# B&R Automation Studio project PP500_1
Automation Studio 4.12.3.127 SP; technology packages: mappCockpit 5.22.0, mappMotion 5.22.0, mappView 5.22.0

## Configuration PP500

CPU 5PP5CP.US15-02, AutomationRuntime F4.83, Build 4.1.2, Safety 1.10, Vc 

### Task classes (Cpu.sw)
```
Cyclic#8 (cycle 9600 us):
  Axis_1 <- Axis_1.prg
  Axis_2 <- Axis_2.prg
DataObjects: McAcpSys
NcDataObjects: McDriveLog
Binaries: arsvcreg, udbdef, mvLoader, McAcpDrv, arflatprv, arcoal, FWRules, TCData, mCoWebSc, McAcpSim, Config_1, ashwac, Settings, User, sysconf, iomap, asfw, arconfig, ashwd, Role, Config_2
Libraries: McBase, MpAxis, McAxis, MpBase, McAcpAx, CoTrace, AsZip, FileIO, runtime, AsSafety, standard, DataObj, AsXml, astime, AsBrStr, arssl, powerlnk, sys_lib, asepl, asieccon
```

### Hardware
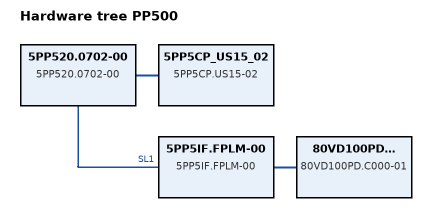
```
5PP520.0702-00 : 5PP520.0702-00 v2.1.3.1
  Connector IF3:
    ActivateDevice = 1
    ActivateSnmp = 2
5PP5CP_US15_02 : 5PP5CP.US15-02 v2.1.6.0  [SY -> 5PP520.0702-00.SY1]
  ConfigurationID = PP500_1_PP500
  UserPartitionSize = 64
  EnableUsbRemoteInstall = 1
  TimerDeviceType = EPLX2X
  TimerDevice = 5PP5IF.FPLM-00.IF1
  TaskClassIdleTime = 1600
  Cyclic1Duration = 800
  Cyclic1Tolerance = 800
  Cyclic3Duration = 40000
  Cyclic3Tolerance = 40000
  Cyclic8Duration = 9600
  FileDevice1
  FileDeviceName1 = USER
  FileDevicePath1 = USER_PATH
  ActivateOpcUa = 1
  OpcUaInformationModels_PV_Version = 1
5PP5IF.FPLM-00 : 5PP5IF.FPLM-00 v2.5.0.0  [SL -> 5PP520.0702-00.SL1]
  Connector IF1:
    CycleTime = 800
80VD100PD.C000-01 : 80VD100PD.C000-01 v2.5.0.0  [PLK1 -> 5PP5IF.FPLM-00.IF1 (NodeNumber=3) [Cable Type=PowerlinkCable, Length=10, Version=1.0.0.3]]
  DriveConfiguration/Module:
    McAcoposTypeID = AcoposMicroDConfig
    ActivateACOPOSSimulationOnPLC = 0
  DriveConfiguration/Channel[1]/RealAxis:
    AxisReference = gAxis_1
    MechanicalElementsIsInvisible = 0
  DriveConfiguration/Channel[1]/RealAxis/MechanicalElements/Gearbox:
    InputIsReadOnly = 0
    Input = 10
    OutputIsReadOnly = 0
    Output = 1
  DriveConfiguration/Channel[1]/RealAxis/MechanicalElements/RotaryToLinearTransformation:
    ReferenceDistanceIsReadOnly = 0
    ReferenceDistance = 36000
  DriveConfiguration/Channel[1]/RealAxis/Controller:
    ModeIsReadOnly = 0
    Mode = PositionControllerWithTorqueFeedForward
  DriveConfiguration/Channel[1]/RealAxis/Controller/Mode/Position:
    ProportionalGainIsReadOnly = 0
    ProportionalGain = 300
    IntegrationTimeIsReadOnly = 0
    IntegrationTime = 0.0
    TotalDelayTime = 0.0004
  DriveConfiguration/Channel[1]/RealAxis/Controller/Mode/Speed:
    ProportionalGainIsReadOnly = 0
    ProportionalGain = 0.4
    IntegrationTimeIsReadOnly = 0
    IntegrationTime = 0.0
    FilterTimeIsReadOnly = 0
    FilterTime = 0.0
  DriveConfiguration/Channel[1]/RealAxis/Controller/Mode:
    FeedForwardIsReadOnly = 0
    FeedForward = Standard
  DriveConfiguration/Channel[1]/RealAxis/Controller/Mode/FeedForward:
    TorqueLoad = 0.0
    TorquePositive = 0.016000
    TorqueNegative = 0.0
    SpeedTorqueFactor = 0.000300
    Inertia = 0.0
    AccelerationFilterTime = 0.0
  DriveConfiguration/Channel[1]/RealAxis/Controller/Mode/LoopFilters:
    LoopFilterXIsReadOnly = 0
    LoopFilter1 = NotUsed
    LoopFilter2 = NotUsed
    LoopFilter3 = NotUsed
  DriveConfiguration/Channel[1]/RealAxis/Homing:
    ModeIsReadOnly = 0
    Mode = Direct
  DriveConfiguration/Channel[1]/RealAxis/Homing/Mode:
    Position = 0.0
    ReferencePulse = NotUsed
  DriveConfiguration/Channel[1]/RealAxis/Homing:
    RestorePositionVariable = 
  DriveConfiguration/Channel[1]/RealAxis/StopReaction:
    QuickstopIsReadOnly = 0
    Quickstop = DecelerationLimit
    DriveErrorIsReadOnly = 0
    DriveError = DecelerationLimit
  DriveConfiguration/Channel[1]/RealAxis/MovementErrorLimits:
    PositionError = 10
    VelocityErrorMonitoring = Automatic1
  DriveConfiguration/Channel[1]/RealAxis:
    JerkFilterIsReadOnly = 0
    JerkFilter = NotUsed
    ZeroVibrationFilter = NotUsed
  DriveConfiguration/Channel[1]/RealAxis/DigitalInputs/HomingSwitch:
    SourceIsReadOnly = 0
    Source = NotUsed
    Level = High
  DriveConfiguration/Channel[1]/RealAxis/DigitalInputs/PositiveLimitSwitch:
    SourceIsReadOnly = 0
    Source = NotUsed
    Level = High
  DriveConfiguration/Channel[1]/RealAxis/DigitalInputs/NegativeLimitSwitch:
    SourceIsReadOnly = 0
    Source = NotUsed
    Level = High
  DriveConfiguration/Channel[1]/RealAxis/DigitalInputs/Trigger1:
    Source = X2Trigger1
    Level = High
  DriveConfiguration/Channel[1]/RealAxis/DigitalInputs/Trigger2:
    Source = X2Trigger2
    Level = High
  DriveConfiguration/Channel[1]/RealAxis/DigitalInputs/Quickstop:
    Input = Trigger2
  DriveConfiguration/Channel[1]/RealAxis/Simulation:
    SimulationModeOnPLC = SetValueGeneration
    SimulationModeOnACOPOS = NotUsed
  DriveConfiguration/Channel[1]/RealAxis/AxisFeatures:
    FeatureRef[1] = AxFeatureBrake
  DriveConfiguration/Channel[2]/RealAxis:
    AxisReference = gAxis_2
    MechanicalElementsIsInvisible = 0
  DriveConfiguration/Channel[2]/RealAxis/MechanicalElements/Gearbox:
    InputIsReadOnly = 0
    Input = 1
    OutputIsReadOnly = 0
    Output = 1
  DriveConfiguration/Channel[2]/RealAxis/MechanicalElements/RotaryToLinearTransformation:
    ReferenceDistanceIsReadOnly = 0
    ReferenceDistance = 36000
  DriveConfiguration/Channel[2]/RealAxis/Controller:
    ModeIsReadOnly = 0
    Mode = PositionController
  DriveConfiguration/Channel[2]/RealAxis/Controller/Mode/Position:
    ProportionalGain = 250
    IntegrationTime = 0.0
    PredictionTime = 0.0004
    TotalDelayTime = 0.0004
  DriveConfiguration/Channel[2]/RealAxis/Controller/Mode/Speed:
    ProportionalGainIsReadOnly = 0
    ProportionalGain = 0.6
    IntegrationTimeIsReadOnly = 0
    IntegrationTime = 0.0
    FilterTimeIsReadOnly = 0
    FilterTime = 0.0
  DriveConfiguration/Channel[2]/RealAxis/Controller/Mode/LoopFilters:
    LoopFilterXIsReadOnly = 0
    LoopFilter1 = NotUsed
    LoopFilter2 = NotUsed
    LoopFilter3 = NotUsed
  DriveConfiguration/Channel[2]/RealAxis/Homing:
    ModeIsReadOnly = 0
    Mode = Direct
  DriveConfiguration/Channel[2]/RealAxis/Homing/Mode:
    Position = 0.0
    ReferencePulse = NotUsed
  DriveConfiguration/Channel[2]/RealAxis/Homing:
    RestorePositionVariable = 
  DriveConfiguration/Channel[2]/RealAxis/StopReaction:
    QuickstopIsReadOnly = 0
    Quickstop = DecelerationLimit
    DriveErrorIsReadOnly = 0
    DriveError = DecelerationLimit
  DriveConfiguration/Channel[2]/RealAxis/MovementErrorLimits:
    PositionError = 1.0
    VelocityErrorMonitoring = Automatic1
  DriveConfiguration/Channel[2]/RealAxis:
    JerkFilterIsReadOnly = 0
    JerkFilter = NotUsed
    ZeroVibrationFilter = NotUsed
  DriveConfiguration/Channel[2]/RealAxis/DigitalInputs/HomingSwitch:
    SourceIsReadOnly = 0
    Source = NotUsed
    Level = High
  DriveConfiguration/Channel[2]/RealAxis/DigitalInputs/PositiveLimitSwitch:
    SourceIsReadOnly = 0
    Source = NotUsed
    Level = High
  DriveConfiguration/Channel[2]/RealAxis/DigitalInputs/NegativeLimitSwitch:
    SourceIsReadOnly = 0
    Source = NotUsed
    Level = High
  DriveConfiguration/Channel[2]/RealAxis/DigitalInputs/Trigger1:
    Source = X2Trigger1
    Level = High
  DriveConfiguration/Channel[2]/RealAxis/DigitalInputs/Trigger2:
    Source = X2Trigger2
    Level = High
  DriveConfiguration/Channel[2]/RealAxis/DigitalInputs/Quickstop:
    Input = Trigger2
  DriveConfiguration/Channel[2]/RealAxis/Simulation:
    SimulationModeOnPLC = SetValueGeneration
    SimulationModeOnACOPOS = NotUsed
```

### Config_1.axis - 5PP5CP_US15_02/mappMotion/Config_1.axis
```
Element gAxis_1 (Type=axis)
  BaseTypeIsReadOnly = 0
  BaseType = Rotary
    MeasurementUnitIsReadOnly = 0
    MeasurementUnit = 17476
    MeasurementResolutionIsReadOnly = 0
    MeasurementResolution = 0.010000
    CountDirectionIsReadOnly = 0
    CountDirection = Standard
  MovementLimitsIsReadOnly = 0
  MovementLimits = Internal
    Position:
      LowerLimitMin = -17976931348623099202083765866295897644998378684266083703805195052047022504132823196914091663318780
      UpperLimitMax = 179769313486230992020837658662958976449983786842660837038051950520470225041328231969140916633187800
      LowerLimit = -1000.000000
      UpperLimit = 1000.000000
    VelocityIsReadOnly = 0
    Velocity:
      VelocityMax = 339999995214436424907732413799364296704.000000
      Velocity = 500
    AccelerationIsReadOnly = 0
    Acceleration:
      AccelerationMax = 339999995214436424907732413799364296704.000000
      Acceleration = 10000
    DecelerationIsReadOnly = 0
    Deceleration:
      DecelerationMax = 339999995214436424907732413799364296704.000000
      Deceleration = 10000
  Alarms = None
```

### Config_2.axis - 5PP5CP_US15_02/mappMotion/Config_2.axis
```
Element gAxis_2 (Type=axis)
  BaseTypeIsReadOnly = 0
  BaseType = Rotary
    MeasurementUnitIsReadOnly = 0
    MeasurementUnit = 17476
    MeasurementResolutionIsReadOnly = 0
    MeasurementResolution = 0.010000
    CountDirectionIsReadOnly = 0
    CountDirection = Standard
  MovementLimitsIsReadOnly = 0
  MovementLimits = Internal
    Position:
      LowerLimitMin = -17976931348623099202083765866295897644998378684266083703805195052047022504132823196914091663318780
      UpperLimitMax = 179769313486230992020837658662958976449983786842660837038051950520470225041328231969140916633187800
      LowerLimit = -1000.000000
      UpperLimit = 1000.000000
    VelocityIsReadOnly = 0
    Velocity:
      VelocityMax = 339999995214436424907732413799364296704.000000
      Velocity = 60000
    AccelerationIsReadOnly = 0
    Acceleration:
      AccelerationMax = 339999995214436424907732413799364296704.000000
      Acceleration = 360000
    DecelerationIsReadOnly = 0
    Deceleration:
      DecelerationMax = 339999995214436424907732413799364296704.000000
      Deceleration = 360000
  Alarms = None
```

### Config_3.axisfeature - 5PP5CP_US15_02/mappMotion/Config_3.axisfeature
```
Element AxFeatureBrake (Type=axisfeature)
  Type = DigitalOutput
    DigitalOutputType = Stepper
      Output = StepperHardware
```

## Logical view

Binary libraries used (declarations not repeated): operator, runtime, astime, AsIecCon, AsZip, FileIO, AsSafety, standard, DataObj, AsXml, AsBrStr, CoTrace 5.24.0, McBase 5.24.0, MpAxis 5.24.0, McAcpAx 5.24.0, McAxis 5.24.0, MpBase

### Package Logical/Libraries - Global libraries

- mCoWebServ.mcowebservercfg (not shown)

### Program Logical/AxisProto (IEC)

#### AxisProtoBrake.typ - Local data types
```iecst
TYPE
	StateOpenCloseEnum :
		(
		STATE_OPEN_CLOSE,
		STATE_STATUS
		);
	AxisBrakeType : 	STRUCT
		CmdClose : BOOL;
		CmdOpen : BOOL;
		CmdSetPar : BOOL;
		ParAxis : McAxisType;
		ParBrake : McAcpAxBrakeParType;
		StaBrake : McBrakeStatusEnum;
		ErrId : DINT;
	END_STRUCT;
END_TYPE
```

#### AxisProtoBrake.var - Local variables
```iecst
(*Axis brake structure, use this structure in your program*)
VAR
	AxisBrake : AxisBrakeType;
END_VAR
(*Local functions and variables*)
VAR
	MC_BR_BrakeSetPar_AcpAx_1 : MC_BR_BrakeSetPar_AcpAx;
	MC_BR_BrakeOperation_1 : MC_BR_BrakeOperation;
	StateOpenClose : StateOpenCloseEnum;
END_VAR
```

#### AxisProtoBrake.st
```iecst
ACTION Brake:
	// --------------------------------------------------------------------------
	// Set brake parameters
	IF AxisBrake.CmdSetPar THEN
		// Preset function block
		MC_BR_BrakeSetPar_AcpAx_1.Execute := 1;
		MC_BR_BrakeSetPar_AcpAx_1.Axis := ADR(AxisBrake.ParAxis);
		MC_BR_BrakeSetPar_AcpAx_1.Parameters := AxisBrake.ParBrake;
		MC_BR_BrakeSetPar_AcpAx_1();

		// Finish when done
		IF MC_BR_BrakeSetPar_AcpAx_1.Done OR MC_BR_BrakeSetPar_AcpAx_1.Error THEN
			// Transfer error id, reset funtion block, reset command
			AxisBrake.ErrId := MC_BR_BrakeSetPar_AcpAx_1.ErrorID;

			MC_BR_BrakeSetPar_AcpAx_1.Execute := 0;
			MC_BR_BrakeSetPar_AcpAx_1();

			AxisBrake.CmdSetPar := FALSE;
		END_IF
	END_IF

	// --------------------------------------------------------------------------
	// Open or close brake
	IF AxisBrake.CmdOpen OR AxisBrake.CmdClose THEN
		CASE StateOpenClose OF
				// --------------------------------------------------------------------------
				// Set brake state
			STATE_OPEN_CLOSE:
				// Preset function block
				MC_BR_BrakeOperation_1.Execute := 1;
				MC_BR_BrakeOperation_1.Axis := ADR(AxisBrake.ParAxis);
				IF AxisBrake.CmdOpen THEN
					MC_BR_BrakeOperation_1.Command := mcBRAKE_OPEN;
				ELSE
					MC_BR_BrakeOperation_1.Command := mcBRAKE_CLOSE;
				END_IF
				MC_BR_BrakeOperation_1();

				// Finish when done
				IF MC_BR_BrakeOperation_1.Done OR MC_BR_BrakeOperation_1.Error THEN
					// Transfer error id, reset funtion block, reset command
					AxisBrake.ErrId := MC_BR_BrakeOperation_1.ErrorID;

					MC_BR_BrakeOperation_1.Execute := 0;
					MC_BR_BrakeOperation_1();

					// Abort when error
					IF MC_BR_BrakeOperation_1.Error THEN
						AxisBrake.CmdOpen := FALSE;
						AxisBrake.CmdClose := FALSE;
					ELSE
						StateOpenClose := STATE_STATUS;
					END_IF
				END_IF
				// --------------------------------------------------------------------------
				// Get brake status
			STATE_STATUS:
				// Preset function block
				MC_BR_BrakeOperation_1.Execute := 1;
				MC_BR_BrakeOperation_1.Axis := ADR(AxisBrake.ParAxis);
				MC_BR_BrakeOperation_1.Command := mcBRAKE_GET_STATUS;
				MC_BR_BrakeOperation_1();

				// Finish when done
				IF MC_BR_BrakeOperation_1.Done OR MC_BR_BrakeOperation_1.Error THEN
					// Transfer error id, status, reset funtion block, reset command
					AxisBrake.ErrId := MC_BR_BrakeOperation_1.ErrorID;
					AxisBrake.StaBrake := MC_BR_BrakeOperation_1.BrakeStatus;

					MC_BR_BrakeOperation_1.Execute := 0;
					MC_BR_BrakeOperation_1();

					AxisBrake.CmdOpen := FALSE;
					AxisBrake.CmdClose := FALSE;

					StateOpenClose := STATE_OPEN_CLOSE;
				END_IF
		END_CASE;

	END_IF

END_ACTION
```

#### AxisProtoParId.typ - Local data types
```iecst
TYPE
	AxisParIdType : 	STRUCT
		CmdSetPar : BOOL;
		CmdGetPar : BOOL;
		ParAxis : McAxisType;
		ParIds : ARRAY[1..AxisParNum]OF McAcpAxProcessParIDType;
		ParNum : UDINT;
		ErrId : DINT;
	END_STRUCT;
END_TYPE
```

#### AxisProtoParId.var - Local variables
```iecst
(*Axis par id structure, use this structure in your program*)
VAR
	AxisParId : AxisParIdType;
END_VAR
(*Local functions and variables*)
VAR
	MC_BR_ProcessParID_AcpAx_1 : MC_BR_ProcessParID_AcpAx;
	mcACPAX_BOOL : ARRAY[1..AxisParNum] OF BOOL;
	mcACPAX_SINT : ARRAY[1..AxisParNum] OF SINT;
	mcACPAX_INT : ARRAY[1..AxisParNum] OF INT;
	mcACPAX_DINT : ARRAY[1..AxisParNum] OF DINT;
	mcACPAX_USINT : ARRAY[1..AxisParNum] OF USINT;
	mcACPAX_UINT : ARRAY[1..AxisParNum] OF UINT;
	mcACPAX_UDINT : ARRAY[1..AxisParNum] OF UDINT;
	mcACPAX_REAL : ARRAY[1..AxisParNum] OF REAL;
END_VAR
(*Configuration*)
VAR CONSTANT
	AxisParNum : USINT := 10;
END_VAR
```

#### AxisProtoParId.st
```iecst
ACTION ParID:
	// Call parameter ID read and write
	IF AxisParId.CmdGetPar OR AxisParId.CmdSetPar THEN
		// Preset function block
		MC_BR_ProcessParID_AcpAx_1.Execute := 1;
		MC_BR_ProcessParID_AcpAx_1.Axis := ADR(AxisParId.ParAxis);
		MC_BR_ProcessParID_AcpAx_1.DataAddress := ADR(AxisParId.ParIds);
		MC_BR_ProcessParID_AcpAx_1.NumberOfParIDs := AxisParId.ParNum;
		IF AxisParId.CmdSetPar THEN
			MC_BR_ProcessParID_AcpAx_1.Mode := mcACPAX_PARID_SET;
		ELSE
			MC_BR_ProcessParID_AcpAx_1.Mode := mcACPAX_PARID_GET;
		END_IF
		MC_BR_ProcessParID_AcpAx_1();

		// Finish when done
		IF MC_BR_ProcessParID_AcpAx_1.Done OR MC_BR_ProcessParID_AcpAx_1.Error THEN
			// Transfer error id, reset funtion block, reset command
			AxisParId.ErrId := MC_BR_ProcessParID_AcpAx_1.ErrorID;

			MC_BR_ProcessParID_AcpAx_1.Execute := 0;
			MC_BR_ProcessParID_AcpAx_1();

			AxisParId.CmdGetPar := FALSE;
			AxisParId.CmdSetPar := FALSE;
		END_IF
	END_IF

	// Avoid compiler warnings
	mcACPAX_BOOL;
	mcACPAX_SINT;
	mcACPAX_INT;
	mcACPAX_DINT;
	mcACPAX_USINT;
	mcACPAX_UINT;
	mcACPAX_UDINT;
	mcACPAX_REAL;
END_ACTION
```

#### AxisProtoAxisCfg.typ - Local data types
```iecst
TYPE
	AxisCfgType : 	STRUCT
		CmdSetAxis : BOOL;
		CmdGetAxis : BOOL;
		CmdReboot : BOOL;
		MpLink : REFERENCE TO McAxisType;
		ParAxis : McCfgAxType;
		StaAxis : McCfgAxType;
		ErrId : DINT;
	END_STRUCT;
	AxisCfgInternalType : 	STRUCT
		ProcessConfig : MC_BR_ProcessConfig;
		GetHardwareInfo : MC_BR_GetHardwareInfo;
		State : AxisCfgStateEnum;
		Name : STRING[32];
		n : UINT;
	END_STRUCT;
	AxisCfgStateEnum :
		(
		STATE_AXIS_CFG_WAIT,
		STATE_AXIS_CFG_PRE_SET,
		STATE_AXIS_CFG_READ,
		STATE_AXIS_CFG_WRITE
		);
END_TYPE
```

#### AxisProtoAxisCfg.st
```iecst
ACTION AxisCfgAction:
	// --------------------------------------------------------------------------
	// Reboot PLC
	IF AxisCfg.CmdReboot THEN
		SYSreset(TRUE, SYSLIB_WARMSTART);
	END_IF

	// --------------------------------------------------------------------------
	// State machine for axis configuration
	CASE AxisCfgInternal.State OF
		// --------------------------------------------------------------------------
		// Wait for new command
		STATE_AXIS_CFG_WAIT:
			IF AxisCfg.CmdGetAxis OR AxisCfg.CmdSetAxis THEN
				// Reset function blocks
				AxisCfgInternal.ProcessConfig.Execute := FALSE;
				AxisCfg.ErrId := ERR_OK;

				AxisCfgInternal.State := STATE_AXIS_CFG_PRE_SET;
			END_IF

		// --------------------------------------------------------------------------
		// Generate address and channel string
		STATE_AXIS_CFG_PRE_SET:
			AxisCfgInternal.GetHardwareInfo.Execute := TRUE;
			AxisCfgInternal.GetHardwareInfo.Axis := AxisCfg.MpLink;

			// Finish when done
			IF AxisCfgInternal.GetHardwareInfo.Done OR AxisCfgInternal.GetHardwareInfo.Error THEN
				// Transfer error id, reset function block
				AxisCfg.ErrId := AxisCfgInternal.GetHardwareInfo.ErrorID;
				AxisCfgInternal.GetHardwareInfo.Execute := FALSE;

				// Abort when error
				IF AxisCfgInternal.GetHardwareInfo.Error THEN
					AxisCfg.CmdSetAxis := FALSE;
					AxisCfg.CmdGetAxis := FALSE;

					AxisCfgInternal.State := STATE_AXIS_CFG_WAIT;
				ELSE
					// Transfer name, read base type first
					AxisCfgInternal.Name := AxisCfgInternal.GetHardwareInfo.HardwareInfo.Axis.AxisName;
					AxisCfgInternal.ProcessConfig.DataType := mcCFG_AX_BASE_TYP;

					// Proceed with command read
					IF AxisCfg.CmdGetAxis THEN
						AxisCfgInternal.ProcessConfig.DataAddress := ADR(AxisCfg.StaAxis.BaseType);
						AxisCfgInternal.State := STATE_AXIS_CFG_READ;
					// Proceed with command write
					ELSE
						AxisCfgInternal.ProcessConfig.DataAddress := ADR(AxisCfg.ParAxis.BaseType);
						AxisCfgInternal.State := STATE_AXIS_CFG_WRITE;
					END_IF
				END_IF
			END_IF

		// --------------------------------------------------------------------------
		// Read Axis data
		STATE_AXIS_CFG_READ:
			// Read Axis configuration
			AxisCfgInternal.ProcessConfig.Execute := TRUE;
			AxisCfgInternal.ProcessConfig.Name := AxisCfgInternal.Name;
			AxisCfgInternal.ProcessConfig.Mode := mcPCM_LOAD;

			// Finish when done
			IF AxisCfgInternal.ProcessConfig.Done OR AxisCfgInternal.ProcessConfig.Error THEN
				// Transfer error id, reset function block
				AxisCfg.ErrId := AxisCfgInternal.ProcessConfig.ErrorID;
				AxisCfgInternal.ProcessConfig.Execute := FALSE;

				// Abort when error
				IF AxisCfgInternal.ProcessConfig.Error THEN
					AxisCfg.CmdSetAxis := FALSE;
					AxisCfg.CmdGetAxis := FALSE;

					AxisCfgInternal.State := STATE_AXIS_CFG_WAIT;
				// Proceed with next step
				ELSE
					// Read movement limits in second run
					IF AxisCfgInternal.ProcessConfig.DataType = mcCFG_AX_BASE_TYP THEN
						AxisCfgInternal.ProcessConfig.DataType := mcCFG_AX_MOVE_LIM;
						AxisCfgInternal.ProcessConfig.DataAddress := ADR(AxisCfg.StaAxis.MovementLimits);
					// Finish command read
					ELSE
						AxisCfg.CmdGetAxis := FALSE;
						AxisCfgInternal.State := STATE_AXIS_CFG_WAIT;
					END_IF
				END_IF
			END_IF

			// --------------------------------------------------------------------------
			// Write axis data
		STATE_AXIS_CFG_WRITE:
			// Read axis configuration
			AxisCfgInternal.ProcessConfig.Execute := TRUE;
			AxisCfgInternal.ProcessConfig.Name := AxisCfgInternal.Name;
			AxisCfgInternal.ProcessConfig.Mode := mcPCM_SAVE;

			// Finish when done
			IF AxisCfgInternal.ProcessConfig.Done OR AxisCfgInternal.ProcessConfig.Error THEN
				// Transfer error id, reset function block
				AxisCfg.ErrId := AxisCfgInternal.ProcessConfig.ErrorID;
				AxisCfgInternal.ProcessConfig.Execute := FALSE;

				// Write movement limits in second run
				IF AxisCfgInternal.ProcessConfig.DataType = mcCFG_AX_BASE_TYP  AND NOT AxisCfgInternal.ProcessConfig.Error THEN
					AxisCfgInternal.ProcessConfig.DataType := mcCFG_AX_MOVE_LIM;
					AxisCfgInternal.ProcessConfig.DataAddress := ADR(AxisCfg.ParAxis.MovementLimits);
				// Finish when done or on error
				ELSE
					AxisCfg.CmdSetAxis := FALSE;
					AxisCfg.CmdGetAxis := FALSE;

					AxisCfgInternal.State := STATE_AXIS_CFG_WAIT;
				END_IF
			END_IF
	END_CASE

	// Cyclic function calls
	AxisCfgInternal.ProcessConfig();
	AxisCfgInternal.GetHardwareInfo();

END_ACTION
```

#### AxisProtoAxisCfg.var - Local variables
```iecst
(*Axis par id structure, use this structure in your program*)
VAR
	AxisCfg : AxisCfgType;
END_VAR
(*Internal structure*)
VAR
	AxisCfgInternal : AxisCfgInternalType;
END_VAR
```

#### AxisConfigSample.st
```iecst
ACTION AxisConfigSample:
	// Axis base type
	AxisCfg.ParAxis.BaseType.Type := mcABT_ROT;
	AxisCfg.ParAxis.BaseType.Rotary.MeasurementResolution := 0.01;
	AxisCfg.ParAxis.BaseType.Rotary.MeasurementUnit := mcCLRU_DEG;
	AxisCfg.ParAxis.BaseType.Rotary.CountDirection := mcCCD_STD;

	// Movement limits
	AxisCfg.ParAxis.MovementLimits.Internal.Acceleration.Basic.Acceleration := 10000;
	AxisCfg.ParAxis.MovementLimits.Internal.Deceleration.Basic.Deceleration := 10000;
	AxisCfg.ParAxis.MovementLimits.Internal.Velocity.Basic.Velocity := 200;

END_ACTION
```

#### revision.txt
```
Version 2
- Renamed function block
- Dont read before write
- Minor tweaks

Version 1
- First release
```

#### AxisProtoBrake.typ - Local data types
```iecst
TYPE
	AxisBrakeType : 	STRUCT
		CmdClose : BOOL;
		CmdOpen : BOOL;
		CmdSetPar : BOOL;
		MpLink : REFERENCE TO McAxisType;
		ParBrake : McAcpAxBrakeParType;
		StaBrake : McBrakeStatusEnum;
		ErrId : DINT;
	END_STRUCT;
	AxisBrakeStateEnum :
		(
		STATE_BRAKE_WAIT,
		STATE_BRAKE_OPEN_CLOSE,
		STATE_BRAKE_STATUS
		);
END_TYPE
```

#### AxisProtoBrake.var - Local variables
```iecst
(*Axis brake structure, use this structure in your program*)
VAR
	AxisBrake : AxisBrakeType;
END_VAR
(*Local functions and variables*)
VAR
	MC_BR_BrakeSetPar_AcpAx_1 : MC_BR_BrakeSetPar_AcpAx;
	MC_BR_BrakeOperation_1 : MC_BR_BrakeOperation;
	AxisBrakeState : AxisBrakeStateEnum;
END_VAR
```

#### AxisProtoBrake.st
```iecst
ACTION AxisBrakeAction:
	// --------------------------------------------------------------------------
	// Set brake parameters
	IF AxisBrake.CmdSetPar THEN
		// Preset function block
		MC_BR_BrakeSetPar_AcpAx_1.Execute := 1;
		MC_BR_BrakeSetPar_AcpAx_1.Axis := AxisBrake.MpLink;
		MC_BR_BrakeSetPar_AcpAx_1.Parameters := AxisBrake.ParBrake;

		// Finish when done
		IF MC_BR_BrakeSetPar_AcpAx_1.Done OR MC_BR_BrakeSetPar_AcpAx_1.Error THEN
			// Transfer error id, reset funtion block, reset command
			AxisBrake.ErrId := MC_BR_BrakeSetPar_AcpAx_1.ErrorID;
			MC_BR_BrakeSetPar_AcpAx_1.Execute := 0;
			AxisBrake.CmdSetPar := FALSE;
		END_IF
	END_IF

	// --------------------------------------------------------------------------
	// Open or close brake
	IF AxisBrake.CmdOpen OR AxisBrake.CmdClose THEN
		CASE AxisBrakeState OF
			// --------------------------------------------------------------------------
			// Wait state
			STATE_BRAKE_WAIT:
				// Command open brake
				IF AxisBrake.CmdOpen THEN
					MC_BR_BrakeOperation_1.Command := mcBRAKE_OPEN;
					AxisBrakeState := STATE_BRAKE_OPEN_CLOSE;
				END_IF

				// Command close brake
				IF AxisBrake.CmdClose THEN
					MC_BR_BrakeOperation_1.Command := mcBRAKE_CLOSE;
					AxisBrakeState := STATE_BRAKE_OPEN_CLOSE;
				END_IF

			// --------------------------------------------------------------------------
			// Set brake state
			STATE_BRAKE_OPEN_CLOSE:
				// Preset function block
				MC_BR_BrakeOperation_1.Execute := TRUE;
				MC_BR_BrakeOperation_1.Axis := AxisBrake.MpLink;

				// Finish when done
				IF MC_BR_BrakeOperation_1.Done OR MC_BR_BrakeOperation_1.Error THEN
					// Transfer error id, reset function block
					AxisBrake.ErrId := MC_BR_BrakeOperation_1.ErrorID;
					MC_BR_BrakeOperation_1.Execute := FALSE;

					// Abort when error
					IF MC_BR_BrakeOperation_1.Error THEN
						AxisBrake.CmdOpen := FALSE;
						AxisBrake.CmdClose := FALSE;

						AxisBrakeState := STATE_BRAKE_WAIT;
					ELSE
						AxisBrakeState := STATE_BRAKE_STATUS;
					END_IF
				END_IF

			// --------------------------------------------------------------------------
			// Get brake status
			STATE_BRAKE_STATUS:
				// Preset function block
				MC_BR_BrakeOperation_1.Execute := 1;
				MC_BR_BrakeOperation_1.Axis := AxisBrake.MpLink;
				MC_BR_BrakeOperation_1.Command := mcBRAKE_GET_STATUS;
				MC_BR_BrakeOperation_1();

				// Finish when done
				IF MC_BR_BrakeOperation_1.Done OR MC_BR_BrakeOperation_1.Error THEN
					// Transfer error id, status, reset funtion block, reset command
					AxisBrake.ErrId := MC_BR_BrakeOperation_1.ErrorID;
					AxisBrake.StaBrake := MC_BR_BrakeOperation_1.BrakeStatus;

					MC_BR_BrakeOperation_1.Execute := 0;

					AxisBrake.CmdOpen := FALSE;
					AxisBrake.CmdClose := FALSE;

					AxisBrakeState := STATE_BRAKE_WAIT;
				END_IF
		END_CASE;
	END_IF

	// Cyclic function calls
	MC_BR_BrakeSetPar_AcpAx_1();
	MC_BR_BrakeOperation_1();

END_ACTION
```

#### revision.txt
```
Version 2
- Renamed action

Version 1
- First release
```

#### AxisProtoCommon.typ - Local data types
```iecst
TYPE
	AxisCommonType : 	STRUCT
		CmdReboot : BOOL;
	END_STRUCT;
END_TYPE
```

#### AxisProtoCommon.var - Local variables
```iecst
(*Generic variables used in multiple actions*)
VAR
	AxisCommon : AxisCommonType;
	n : UINT;
END_VAR
```

#### AxisProtoCommon.st
```iecst
ACTION AxisCommonAction:
	// --------------------------------------------------------------------------
	// Reboot PLC
	IF AxisCommon.CmdReboot THEN
		SYSreset(TRUE, SYSLIB_WARMSTART);
	END_IF

	// --------------------------------------------------------------------------
	// Avoid compiler warnings
	n;

END_ACTION
```

#### revision.txt
```
Version 3
- Renamed action
- Avoid compiler warnings

Version 2
- Renamed action

Version 1
- First release
```

#### AxisProtoDriveCfg.typ - Local data types
```iecst
TYPE
	AxisDriveCfgType : 	STRUCT
		CmdSetDrive : BOOL;
		CmdGetDrive : BOOL;
		CmdReboot : BOOL;
		MpLink : REFERENCE TO McAxisType;
		ParDrive : McCfgAcpAxType;
		StaDrive : McCfgAcpAxType;
		ErrId : DINT;
	END_STRUCT;
	AxisDriveCfgInternalType : 	STRUCT
		ProcessConfig : MC_BR_ProcessConfig;
		GetHardwareInfo : MC_BR_GetHardwareInfo;
		State : AxisDriveCfgStateEnum;
		Address : STRING[64];
		Channel : STRING[64];
		myFeatures : ARRAY[0..8]OF McCfgReferenceType;
		n : UINT;
	END_STRUCT;
	AxisDriveCfgStateEnum :
		(
		STATE_DRIVE_CFG_WAIT,
		STATE_DRIVE_CFG_PRE_SET,
		STATE_DRIVE_CFG_READ,
		STATE_DRIVE_CFG_WRITE
		);
END_TYPE
```

#### AxisProtoDriveCfg.var - Local variables
```iecst
(*Axis par id structure, use this structure in your program*)
VAR
	AxisDriveCfg : AxisDriveCfgType;
END_VAR
(*Internal structure*)
VAR
	AxisDriveCfgInternal : AxisDriveCfgInternalType;
END_VAR
(*Generic error numbers*)
VAR
	ERR_AXISDRIVECFG_LOC_EMPTY : UINT := 10000; (*Axis location is empty*)
	ERR_AXISDRIVECFG_LOC_INVALID : UINT := 10001; (*Axis location is invalid*)
	ERR_AXISDRIVECFG_AX_FEATURE : UINT := 10002; (*Axis feature configuration is invalid*)
END_VAR
```

#### AxisProtoDriveCfg.st
```iecst
ACTION AxisDriveCfgAction:
	// --------------------------------------------------------------------------
	// Reboot PLC
	IF AxisDriveCfg.CmdReboot THEN
		SYSreset(TRUE, SYSLIB_WARMSTART);
	END_IF

	// --------------------------------------------------------------------------
	// State machine for axis configuration
	CASE AxisDriveCfgInternal.State OF
		// --------------------------------------------------------------------------
		// Wait for new command
		STATE_DRIVE_CFG_WAIT:
			// Command read configuration
			IF AxisDriveCfg.CmdGetDrive THEN
				// Reset function blocks and erros
				AxisDriveCfgInternal.ProcessConfig.Execute := FALSE;
				AxisDriveCfg.ErrId := ERR_OK;

				// Make correction for axis feature
				IF AxisDriveCfg.StaDrive.AxisFeatures.FeatureReference.DataAddress = 0 THEN
					AxisDriveCfg.StaDrive.AxisFeatures.FeatureReference.DataAddress := ADR(AxisDriveCfgInternal.myFeatures);
					AxisDriveCfg.StaDrive.AxisFeatures.FeatureReference.NumberOfArrayElements := SIZEOF(AxisDriveCfgInternal.myFeatures)/SIZEOF(AxisDriveCfgInternal.myFeatures[0]);
				END_IF

				AxisDriveCfgInternal.State := STATE_DRIVE_CFG_PRE_SET;
			END_IF

			// Command write configuration
			IF AxisDriveCfg.CmdSetDrive THEN
				// Make axis feature has valid pointer
				IF AxisDriveCfg.StaDrive.AxisFeatures.FeatureReference.DataAddress = 0 AND AxisDriveCfg.StaDrive.AxisFeatures.FeatureReference.NumberOfElements > 0 THEN
					AxisDriveCfg.ErrId := ERR_AXISDRIVECFG_AX_FEATURE;
					AxisDriveCfg.CmdSetDrive := 0;
				ELSE
					// Reset function blocks and erros
					AxisDriveCfgInternal.ProcessConfig.Execute := FALSE;
					AxisDriveCfg.ErrId := ERR_OK;

					AxisDriveCfgInternal.State := STATE_DRIVE_CFG_PRE_SET;
				END_IF

			END_IF

		// --------------------------------------------------------------------------
		// Generate address and channel string
		STATE_DRIVE_CFG_PRE_SET:
			AxisDriveCfgInternal.GetHardwareInfo.Execute := TRUE;
			AxisDriveCfgInternal.GetHardwareInfo.Axis := AxisDriveCfg.MpLink;

			// Finish when done
			IF AxisDriveCfgInternal.GetHardwareInfo.Done OR AxisDriveCfgInternal.GetHardwareInfo.Error THEN
				// Transfer error id, reset function block
				AxisDriveCfg.ErrId := AxisDriveCfgInternal.GetHardwareInfo.ErrorID;
				AxisDriveCfgInternal.GetHardwareInfo.Execute := FALSE;

				// Abort when error or command was read
				IF AxisDriveCfgInternal.GetHardwareInfo.Error THEN
					AxisDriveCfg.CmdSetDrive := FALSE;
					AxisDriveCfg.CmdGetDrive := FALSE;

					AxisDriveCfgInternal.State := STATE_DRIVE_CFG_WAIT;
				ELSE
					// Make sure location is not empty
					IF AxisDriveCfgInternal.GetHardwareInfo.HardwareInfo.Axis.ConfigElementLocation <> '' THEN
						// Extract location string
						AxisDriveCfgInternal.n := FIND(AxisDriveCfgInternal.GetHardwareInfo.HardwareInfo.Axis.ConfigElementLocation, '/');
						IF AxisDriveCfgInternal.n > 0 THEN
							AxisDriveCfgInternal.Address := LEFT(AxisDriveCfgInternal.GetHardwareInfo.HardwareInfo.Axis.ConfigElementLocation, AxisDriveCfgInternal.n - 1);
							AxisDriveCfgInternal.Channel := RIGHT(AxisDriveCfgInternal.GetHardwareInfo.HardwareInfo.Axis.ConfigElementLocation, 8);
							IF AxisDriveCfgInternal.Channel = 'Channel1' THEN
								AxisDriveCfgInternal.Address := CONCAT(AxisDriveCfgInternal.Address, '/DriveConfiguration/Channel1');
							ELSIF AxisDriveCfgInternal.Channel = 'Channel2' THEN
								AxisDriveCfgInternal.Address := CONCAT(AxisDriveCfgInternal.Address, '/DriveConfiguration/Channel2');
							ELSE
								AxisDriveCfgInternal.Address := CONCAT(AxisDriveCfgInternal.Address, '/DriveConfiguration/Channel3');
							END_IF

							// Proceed with command is get
							IF AxisDriveCfg.CmdGetDrive THEN
								AxisDriveCfgInternal.State := STATE_DRIVE_CFG_READ;
								// Proceed with command is set
							ELSE
								AxisDriveCfgInternal.State := STATE_DRIVE_CFG_WRITE;
							END_IF
							// Cannot extract location string
						ELSE
							AxisDriveCfg.ErrId := ERR_AXISDRIVECFG_LOC_INVALID;
							AxisDriveCfg.CmdSetDrive := FALSE;
							AxisDriveCfg.CmdGetDrive := FALSE;
							AxisDriveCfgInternal.State := STATE_DRIVE_CFG_WAIT;
						END_IF
						// Location is not empty
					ELSE
						AxisDriveCfg.ErrId := ERR_AXISDRIVECFG_LOC_EMPTY;
						AxisDriveCfg.CmdSetDrive := FALSE;
						AxisDriveCfg.CmdGetDrive := FALSE;
						AxisDriveCfgInternal.State := STATE_DRIVE_CFG_WAIT;
					END_IF
				END_IF
			END_IF

		// --------------------------------------------------------------------------
		// Read drive data
		STATE_DRIVE_CFG_READ:
			// Read Axis configuration
			AxisDriveCfgInternal.ProcessConfig.Execute := TRUE;
			AxisDriveCfgInternal.ProcessConfig.Name := AxisDriveCfgInternal.Address;
			AxisDriveCfgInternal.ProcessConfig.DataType := mcCFG_ACP_AX;
			AxisDriveCfgInternal.ProcessConfig.DataAddress := ADR(AxisDriveCfg.StaDrive);
			AxisDriveCfgInternal.ProcessConfig.Mode := mcPCM_LOAD;

			// Finish when done
			IF AxisDriveCfgInternal.ProcessConfig.Done OR AxisDriveCfgInternal.ProcessConfig.Error THEN
				// Transfer error id, reset function block
				AxisDriveCfg.ErrId := AxisDriveCfgInternal.ProcessConfig.ErrorID;
				AxisDriveCfgInternal.ProcessConfig.Execute := FALSE;
				AxisDriveCfg.CmdGetDrive := FALSE;

				AxisDriveCfgInternal.State := STATE_DRIVE_CFG_WAIT;
			END_IF

		// --------------------------------------------------------------------------
		// Write drive data
		STATE_DRIVE_CFG_WRITE:
			// Read axis configuration
			AxisDriveCfgInternal.ProcessConfig.Execute := TRUE;
			AxisDriveCfgInternal.ProcessConfig.Name := AxisDriveCfgInternal.Address;
			AxisDriveCfgInternal.ProcessConfig.DataType := mcCFG_ACP_AX;
			AxisDriveCfgInternal.ProcessConfig.DataAddress := ADR(AxisDriveCfg.ParDrive);
			AxisDriveCfgInternal.ProcessConfig.Mode := mcPCM_SAVE;

			// Finish when done
			IF AxisDriveCfgInternal.ProcessConfig.Done OR AxisDriveCfgInternal.ProcessConfig.Error THEN
				// Transfer error id, reset function block
				AxisDriveCfg.ErrId := AxisDriveCfgInternal.ProcessConfig.ErrorID;
				AxisDriveCfgInternal.ProcessConfig.Execute := FALSE;
				AxisDriveCfg.CmdSetDrive := FALSE;

				AxisDriveCfgInternal.State := STATE_DRIVE_CFG_WAIT;
			END_IF
	END_CASE

	// --------------------------------------------------------------------------
	// Cyclic function calls
	AxisDriveCfgInternal.ProcessConfig();
	AxisDriveCfgInternal.GetHardwareInfo();

END_ACTION
```

#### DriveConfigSample.st
```iecst
ACTION AxisConfigSample:
	// Drive controller configuration
	AxisDriveCfg.ParDrive.Controller.Mode.PositionControllerTorqueFf.Position.ProportionalGain := 200;
	AxisDriveCfg.ParDrive.Controller.Mode.PositionControllerTorqueFf.Position.IntegrationTime := 0;
	AxisDriveCfg.ParDrive.Controller.Mode.PositionControllerTorqueFf.Position.TotalDelayTime := 0.0004;

END_ACTION
```

#### revision.txt
```
Version 3
- Update mappMotion to 5.24
- Removed obsolete hardware
- Added axis feature pointer auto correction

Version 2
- Removed dependency from common
- New internal structure

Version 1
- First release
```

#### AxisProtoGlobal.var - Local variables
```iecst
(*Generic variables used in multiple actions*)
VAR
	n : UINT;
END_VAR
```

#### AxisProtoMotorCfg.typ - Local data types
```iecst
TYPE
	AxisMotorCfgType : 	STRUCT
		CmdSetMotor : BOOL;
		CmdGetMotor : BOOL;
		CmdReboot : BOOL;
		MpLink : REFERENCE TO McAxisType;
		ParMotorType : UDINT;
		ParMotorSynchronous : McCfgMotSynType;
		StaMotorSynchronous : McCfgMotSynType;
		ParMotorInduction : McCfgMotInductType;
		StaMotorInduction : McCfgMotInductType;
		StaCompareResult : BOOL;
		ErrId : DINT;
	END_STRUCT;
	AxisMotorCfgInternalType : 	STRUCT
		ProcessConfig : MC_BR_ProcessConfig;
		GetHardwareInfo : MC_BR_GetHardwareInfo;
		State : AxisMotorCfgStateEnum;
		Address : STRING[32];
		Channel : STRING[32];
		n : UINT;
	END_STRUCT;
	AxisMotorCfgTypeEnum :
		(
		AX_MOTOR_TYPE_UNDEFINED,
		AX_MOTOR_TYPE_SYNCHRONOUS,
		AX_MOTOR_TYPE_INDUCTION
		);
	AxisMotorCfgStateEnum :
		(
		STATE_MOTOR_CFG_WAIT,
		STATE_MOTOR_CFG_PRE_SET,
		STATE_MOTOR_CFG_READ,
		STATE_MOTOR_CFG_WRITE
		);
END_TYPE
```

#### AxisProtoMotorCfg.var - Local variables
```iecst
(*Axis par id structure, use this structure in your program*)
VAR
	AxisMotorCfg : AxisMotorCfgType;
END_VAR
(*Internal variables*)
VAR
	AxisMotorCfgInternal : AxisMotorCfgInternalType;
END_VAR
(*Local Errors*)
VAR
	ERR_AXISMOTORCFG_LOC_EMPTY : UINT := 10000; (*Axis location is empty*)
	ERR_AXISMOTORCFG_LOC_INVALID : UINT := 10001;
END_VAR
```

#### AxisProtoMotorCfg.st
```iecst
ACTION MotorCfgAction:
	// --------------------------------------------------------------------------
	// Reboot PLC
	IF AxisMotorCfg.CmdReboot THEN
		SYSreset(TRUE, SYSLIB_WARMSTART);
	END_IF

	// --------------------------------------------------------------------------
	// State machine for motor configuration
	CASE AxisMotorCfgInternal.State OF
		// --------------------------------------------------------------------------
		// Wait for new command
		STATE_MOTOR_CFG_WAIT:
			IF AxisMotorCfg.CmdGetMotor OR AxisMotorCfg.CmdSetMotor THEN
				// Reset function blocks and errors
				AxisMotorCfgInternal.ProcessConfig.Execute := FALSE;
				AxisMotorCfg.ErrId := ERR_OK;

				AxisMotorCfgInternal.State := STATE_MOTOR_CFG_PRE_SET;
			END_IF

			// --------------------------------------------------------------------------
			// Generate address and channel string
		STATE_MOTOR_CFG_PRE_SET:
			AxisMotorCfgInternal.GetHardwareInfo.Execute := TRUE;
			AxisMotorCfgInternal.GetHardwareInfo.Axis := AxisMotorCfg.MpLink;

			// Finish when done
			IF AxisMotorCfgInternal.GetHardwareInfo.Done OR AxisMotorCfgInternal.GetHardwareInfo.Error THEN
				// Transfer error id, reset function block
				AxisMotorCfg.ErrId := AxisMotorCfgInternal.GetHardwareInfo.ErrorID;
				AxisMotorCfgInternal.GetHardwareInfo.Execute := FALSE;

				// Abort when error or command was read
				IF AxisMotorCfgInternal.GetHardwareInfo.Error THEN
					AxisMotorCfg.CmdSetMotor := FALSE;
					AxisMotorCfg.CmdGetMotor := FALSE;

					AxisMotorCfgInternal.State := STATE_MOTOR_CFG_WAIT;
				ELSE
					// Make sure location is not empty
					IF AxisMotorCfgInternal.GetHardwareInfo.HardwareInfo.Axis.ConfigElementLocation <> '' THEN
						// Extract location string
						AxisMotorCfgInternal.n := FIND(AxisMotorCfgInternal.GetHardwareInfo.HardwareInfo.Axis.ConfigElementLocation, '/');
						IF AxisMotorCfgInternal.n > 0 THEN
							AxisMotorCfgInternal.Address := LEFT(AxisMotorCfgInternal.GetHardwareInfo.HardwareInfo.Axis.ConfigElementLocation, AxisMotorCfgInternal.n - 1);
							AxisMotorCfgInternal.Channel := RIGHT(AxisMotorCfgInternal.GetHardwareInfo.HardwareInfo.Axis.ConfigElementLocation, 8);
							IF AxisMotorCfgInternal.Channel = 'Channel1' THEN
								AxisMotorCfgInternal.Address := CONCAT(AxisMotorCfgInternal.Address, '.M1/M1');
							ELSIF AxisMotorCfgInternal.Channel = 'Channel2' THEN
								AxisMotorCfgInternal.Address := CONCAT(AxisMotorCfgInternal.Address, '.M2/M1');
							ELSE
								AxisMotorCfgInternal.Address := CONCAT(AxisMotorCfgInternal.Address, '.M3/M1');
							END_IF

							// Procced with command read
							IF AxisMotorCfg.CmdGetMotor THEN
								AxisMotorCfgInternal.State := STATE_MOTOR_CFG_READ;
								// Procced with command write
							ELSE
								AxisMotorCfgInternal.State := STATE_MOTOR_CFG_WRITE;
							END_IF
							// Cannot extract location string
						ELSE
							AxisMotorCfg.ErrId := ERR_AXISMOTORCFG_LOC_INVALID;
							AxisMotorCfg.CmdSetMotor := FALSE;
							AxisMotorCfg.CmdGetMotor := FALSE;
							AxisMotorCfgInternal.State := STATE_MOTOR_CFG_WAIT;
						END_IF
						// Location is not empty
					ELSE
						AxisMotorCfg.ErrId := ERR_AXISMOTORCFG_LOC_EMPTY;
						AxisMotorCfg.CmdSetMotor := FALSE;
						AxisMotorCfg.CmdGetMotor := FALSE;
						AxisMotorCfgInternal.State := STATE_MOTOR_CFG_WAIT;
					END_IF
				END_IF
			END_IF

			// --------------------------------------------------------------------------
			// Read motor data
		STATE_MOTOR_CFG_READ:
			// Read motor configuration
			AxisMotorCfgInternal.ProcessConfig.Execute := TRUE;
			AxisMotorCfgInternal.ProcessConfig.Name := AxisMotorCfgInternal.Address;
			IF AxisMotorCfg.ParMotorType = AX_MOTOR_TYPE_SYNCHRONOUS THEN
				AxisMotorCfgInternal.ProcessConfig.DataAddress := ADR(AxisMotorCfg.StaMotorSynchronous);
				AxisMotorCfgInternal.ProcessConfig.DataType := mcCFG_MOT_SYN;
			ELSE
				AxisMotorCfgInternal.ProcessConfig.DataAddress := ADR(AxisMotorCfg.StaMotorInduction);
				AxisMotorCfgInternal.ProcessConfig.DataType := mcCFG_MOT_INDUCT;
			END_IF
			AxisMotorCfgInternal.ProcessConfig.Mode := mcPCM_LOAD;

			// Finish when done
			IF AxisMotorCfgInternal.ProcessConfig.Done OR AxisMotorCfgInternal.ProcessConfig.Error THEN
				// Check if Par and Sta structures are identical
				IF AxisMotorCfg.ParMotorType = AX_MOTOR_TYPE_SYNCHRONOUS THEN
					AxisMotorCfg.StaCompareResult := NOT DINT_TO_BOOL(brsmemcmp(ADR(AxisMotorCfg.StaMotorSynchronous), ADR(AxisMotorCfg.ParMotorSynchronous), SIZEOF(AxisMotorCfg.StaMotorSynchronous)));
				ELSE
					AxisMotorCfg.StaCompareResult := NOT DINT_TO_BOOL(brsmemcmp(ADR(AxisMotorCfg.StaMotorInduction), ADR(AxisMotorCfg.ParMotorInduction), SIZEOF(AxisMotorCfg.StaMotorInduction)));
				END_IF

				// Transfer error id, reset function block
				AxisMotorCfg.ErrId := AxisMotorCfgInternal.ProcessConfig.ErrorID;
				AxisMotorCfgInternal.ProcessConfig.Execute := FALSE;

				AxisMotorCfg.CmdSetMotor := FALSE;
				AxisMotorCfg.CmdGetMotor := FALSE;

				AxisMotorCfgInternal.State := STATE_MOTOR_CFG_WAIT;
			END_IF

			// --------------------------------------------------------------------------
			// Write motor data
		STATE_MOTOR_CFG_WRITE:
			// Read motor configuration
			AxisMotorCfgInternal.ProcessConfig.Execute := TRUE;
			AxisMotorCfgInternal.ProcessConfig.Name := AxisMotorCfgInternal.Address;
			IF AxisMotorCfg.ParMotorType = AX_MOTOR_TYPE_SYNCHRONOUS THEN
				AxisMotorCfgInternal.ProcessConfig.DataAddress := ADR(AxisMotorCfg.ParMotorSynchronous);
				AxisMotorCfgInternal.ProcessConfig.DataType := mcCFG_MOT_SYN;
			ELSE
				AxisMotorCfgInternal.ProcessConfig.DataAddress := ADR(AxisMotorCfg.ParMotorInduction);
				AxisMotorCfgInternal.ProcessConfig.DataType := mcCFG_MOT_INDUCT;
			END_IF
			AxisMotorCfgInternal.ProcessConfig.Mode := mcPCM_SAVE;

			// Finish when done
			IF AxisMotorCfgInternal.ProcessConfig.Done OR AxisMotorCfgInternal.ProcessConfig.Error THEN
				// Transfer error id, reset function block
				AxisMotorCfg.ErrId := AxisMotorCfgInternal.ProcessConfig.ErrorID;
				AxisMotorCfgInternal.ProcessConfig.Execute := FALSE;

				AxisMotorCfg.CmdSetMotor := FALSE;
				AxisMotorCfg.CmdGetMotor := FALSE;

				AxisMotorCfgInternal.State := STATE_MOTOR_CFG_WAIT;
			END_IF
	END_CASE

	// Cyclic function calls
	AxisMotorCfgInternal.ProcessConfig();
	AxisMotorCfgInternal.GetHardwareInfo();
END_ACTION
```

#### Motor_8LVB13_B1030F300_00.st
```iecst
ACTION Motor_8LVB13_B1030F300_00:
	// Winding data
	AxisMotorCfg.ParMotorSynchronous.Motor.Type := mcMSM_DEF;
	AxisMotorCfg.ParMotorSynchronous.Motor.Default.NumberOfPolePairs := 4;
	AxisMotorCfg.ParMotorSynchronous.Motor.Default.NominalSpeed := 3000.0;
	AxisMotorCfg.ParMotorSynchronous.Motor.Default.MaximumSpeed := 6600.0;
	AxisMotorCfg.ParMotorSynchronous.Motor.Default.NominalVoltage := 57.0;
	AxisMotorCfg.ParMotorSynchronous.Motor.Default.NominalCurrent := 1.4;
	AxisMotorCfg.ParMotorSynchronous.Motor.Default.StallCurrent := 1.6;
	AxisMotorCfg.ParMotorSynchronous.Motor.Default.PeakCurrent := 5.2;
	AxisMotorCfg.ParMotorSynchronous.Motor.Default.NominalTorque := 0.32;
	AxisMotorCfg.ParMotorSynchronous.Motor.Default.StallTorque := 0.36;
	AxisMotorCfg.ParMotorSynchronous.Motor.Default.PeakTorque := 1;
	AxisMotorCfg.ParMotorSynchronous.Motor.Default.VoltageConstant := 13.61;
	AxisMotorCfg.ParMotorSynchronous.Motor.Default.TorqueConstant := 0.23;
	AxisMotorCfg.ParMotorSynchronous.Motor.Default.StatorResistance := 5.8;
	AxisMotorCfg.ParMotorSynchronous.Motor.Default.StatorInductance := 10.2;
	AxisMotorCfg.ParMotorSynchronous.Motor.Default.MomentOfInertia := 0.03;
	AxisMotorCfg.ParMotorSynchronous.Motor.Default.NominalAmbientTemperature := 40.0;
	// Voltage limitation
	AxisMotorCfg.ParMotorSynchronous.Motor.Default.VoltageLimitation.Type := mcMSMDVL_USE;
	AxisMotorCfg.ParMotorSynchronous.Motor.Default.VoltageLimitation.Used.MaximumDCBusVoltage := 450.0;
	// encoder mounting
	AxisMotorCfg.ParMotorSynchronous.Motor.Default.EncoderMounting.Angle.Type := mcMSMDEMA_VAL_STO_ON_ENC;
	AxisMotorCfg.ParMotorSynchronous.Motor.Default.EncoderMounting.Angle.UserDefined.CommutationOffset := 0.0;
	AxisMotorCfg.ParMotorSynchronous.Motor.Default.EncoderMounting.Angle.Undefined.AutomaticIdentification.Type := mcMSMDEMAUAI_NOT_USE;
	// Temperature sensor
	AxisMotorCfg.ParMotorSynchronous.Motor.Default.TemperatureSensor.Type := mcMMTS_NOT_USE;
	// Temperature model
	AxisMotorCfg.ParMotorSynchronous.Motor.Default.TemperatureModel.Type := mcMMTM_CUR_AND_SPDBASED;
	AxisMotorCfg.ParMotorSynchronous.Motor.Default.TemperatureModel.CurrentAndSpeedBased.LimitTemperature := 110.0;
	AxisMotorCfg.ParMotorSynchronous.Motor.Default.TemperatureModel.CurrentAndSpeedBased.CalculationMethod.Type := mcMMTMCSBCM_SECORD_THRM_NETW;
	AxisMotorCfg.ParMotorSynchronous.Motor.Default.TemperatureModel.CurrentAndSpeedBased.CalculationMethod.SecondOrderThermalNetwork.WindingCrossSection := 0.135;
	AxisMotorCfg.ParMotorSynchronous.Motor.Default.TemperatureModel.CurrentAndSpeedBased.CalculationMethod.SecondOrderThermalNetwork.ThermalTimeConstant := 900.0;
	AxisMotorCfg.ParMotorSynchronous.Motor.Default.TemperatureModel.CurrentAndSpeedBased.CalculationMethod.SecondOrderThermalNetwork.ReferenceTemperature.Type := mcMMTMCSBCMRT_NOM_AMB_TMP;
	// Brake
	AxisMotorCfg.ParMotorSynchronous.Brake.Type := mcMSB_USE;
	AxisMotorCfg.ParMotorSynchronous.Brake.Used.NominalCurrent := 0.33;
	AxisMotorCfg.ParMotorSynchronous.Brake.Used.NominalTorque := 0.35;
	AxisMotorCfg.ParMotorSynchronous.Brake.Used.ActivationDelay := 0.01;
	AxisMotorCfg.ParMotorSynchronous.Brake.Used.ReleaseDelay := 0.006;
	AxisMotorCfg.ParMotorSynchronous.Brake.Used.MomentOfInertia := 0.013;
	AxisMotorCfg.ParMotorSynchronous.Brake.Used.ControlMode.Type := mcMSBUCM_SW;
	// Encoder
	AxisMotorCfg.ParMotorSynchronous.Encoder.Type := mcMSE_USE;
	AxisMotorCfg.ParMotorSynchronous.Encoder.Used.MomentOfInertia := 0.0014;
	AxisMotorCfg.ParMotorSynchronous.Encoder.Used.TemperatureSensor.Type := mcMSEUTS_NOT_USE;
	// Gear box
	AxisMotorCfg.ParMotorSynchronous.Gearbox.Type := mcMSG_NOT_USE;
END_ACTION
```

#### revision.txt
```
Version 6
- Update to mapp 5.23

Version 5
- New flag StaCompareResult shows if parameters in Sta... and Par... are identical

Version 4
- Removed dependency from common
- New internal structure

Version 3
- Renamed function block
- Dont read before write
- Minor tweaks

Version 2
- Renamed action

Version 1
- First release
```

#### AxisProtoParId.typ - Local data types
```iecst
TYPE
	AxisParIdModeType :
		(
		mcACPAX_PARID_DONE,
		mcACPAX_PARID_GET_ONCE,
		mcACPAX_PARID_SET_ONCE,
		mcACPAX_PARID_GET_CYCLIC,
		mcACPAX_PARID_SET_CYCLIC,
		mcACPAX_PARID_GET_MULTI,
		mcACPAX_PARID_SET_MULTI
		);
	AxisParIdInternalType : 	STRUCT
		ProcessParIDGet : MC_BR_ProcessParID_AcpAx;
		ProcessParIDSet : MC_BR_ProcessParID_AcpAx;
		CyclicProcessParIDGet : MC_BR_CyclicProcessParID_AcpAx;
		CyclicProcessParIDSet : MC_BR_CyclicProcessParID_AcpAx;
		GetCyclicDataInfo : MC_BR_GetCyclicDataInfo_AcpAx;
		DataOnceGet : ARRAY[1..AxisParNum]OF McAcpAxProcessParIDType;
		DataOnceSet : ARRAY[1..AxisParNum]OF McAcpAxProcessParIDType;
		DataCylicGet : ARRAY[1..AxisParNum]OF McAcpAxCycParIDType;
		DataCylicSet : ARRAY[1..AxisParNum]OF McAcpAxCycParIDType;
		DataOnceGetIdx : USINT;
		DataOnceSetIdx : USINT;
		DataCyclicGetIdx : USINT;
		DataCyclicSetIdx : USINT;
		VariableStatus : UINT;
		VariableType : UDINT;
		VariableAdr : UDINT;
		VariableLen : UDINT;
		VariableDimension : UDINT;
		McVariableType : ARRAY[1..AxisParNum]OF UDINT;
		McVariableAdr : ARRAY[1..AxisParNum]OF UDINT;
		n : UINT;
		m : UINT;
	END_STRUCT;
	AxisParIdDataType : 	STRUCT
		Execute : AxisParIdModeType;
		ParID : UINT;
		Variable : STRING[250];
	END_STRUCT;
	AxisParIdType : 	STRUCT
		CmdUpdate : BOOL;
		MpLink : REFERENCE TO McAxisType;
		ParIds : ARRAY[1..AxisParNum]OF AxisParIdDataType;
		MaxWriteDataBytes : USINT;
		MaxReadDataBytes : USINT;
		ErrId : DINT;
	END_STRUCT;
END_TYPE
```

#### AxisProtoParId.var - Local variables
```iecst
(*Axis par id structure, use this structure in your program*)
VAR
	AxisParId : AxisParIdType;
END_VAR
(*Local functions and variables*)
VAR
	AxisParIdInternal : AxisParIdInternalType;
END_VAR
(*Configuration*)
VAR CONSTANT
	AxisParNum : USINT := 20;
END_VAR
```

#### AxisProtoParId.st
```iecst
ACTION ParIDAction:
	// --------------------------------------------------------------------------
	// Update configuration data
	IF EDGEPOS(AxisParId.CmdUpdate) THEN
		// Reset counter, internal queue and function block
		AxisParId.ErrId := 0;

		AxisParIdInternal.DataCyclicGetIdx := 0;
		AxisParIdInternal.DataCyclicSetIdx := 0;
		brsmemset(ADR(AxisParIdInternal.DataCylicGet), 0, SIZEOF(AxisParIdInternal.DataCylicGet));
		brsmemset(ADR(AxisParIdInternal.DataCylicSet), 0, SIZEOF(AxisParIdInternal.DataCylicSet));

		AxisParIdInternal.CyclicProcessParIDGet.Enable := FALSE;
		AxisParIdInternal.CyclicProcessParIDGet();
		AxisParIdInternal.CyclicProcessParIDSet.Enable := FALSE;
		AxisParIdInternal.CyclicProcessParIDSet();
		AxisParIdInternal.GetCyclicDataInfo.Execute := FALSE;
		AxisParIdInternal.GetCyclicDataInfo();
	END_IF

	// --------------------------------------------------------------------------
	// Create get once queue
	IF AxisParIdInternal.DataOnceGetIdx = 0  THEN
		FOR AxisParIdInternal.n:=1 TO AxisParNum DO
			// Transfer get once data
			IF AxisParId.ParIds[AxisParIdInternal.n].Execute = mcACPAX_PARID_GET_ONCE THEN
				AxisParIdInternal.DataOnceGetIdx := AxisParIdInternal.DataOnceGetIdx + 1;
				GetVarData;
				// Variable data is valid
				IF AxisParIdInternal.VariableStatus = 0 THEN
					AxisParIdInternal.DataOnceGet[AxisParIdInternal.DataOnceGetIdx].ParID := AxisParId.ParIds[AxisParIdInternal.n].ParID;
					AxisParIdInternal.DataOnceGet[AxisParIdInternal.DataOnceGetIdx].VariableAddress := AxisParIdInternal.McVariableAdr[AxisParIdInternal.n];
					AxisParIdInternal.DataOnceGet[AxisParIdInternal.DataOnceGetIdx].DataType := AxisParIdInternal.McVariableType[AxisParIdInternal.n];
				// Error reading variable data
				ELSE
					AxisParId.ErrId := AxisParIdInternal.VariableStatus;
					AxisParId.ParIds[AxisParIdInternal.n].Execute := mcACPAX_PARID_DONE;
				END_IF
			END_IF
		END_FOR;
	END_IF

	// --------------------------------------------------------------------------
	// Execute get once queue
	IF AxisParIdInternal.DataOnceGetIdx > 0 THEN
		// Preset function block
		AxisParIdInternal.ProcessParIDGet.Execute := 1;
		AxisParIdInternal.ProcessParIDGet.Axis := AxisParId.MpLink;
		AxisParIdInternal.ProcessParIDGet.DataAddress := ADR(AxisParIdInternal.DataOnceGet);
		AxisParIdInternal.ProcessParIDGet.NumberOfParIDs := AxisParIdInternal.DataOnceGetIdx;
		AxisParIdInternal.ProcessParIDGet.Mode := mcACPAX_PARID_GET;

		// Finish when done
		IF AxisParIdInternal.ProcessParIDGet.Done OR AxisParIdInternal.ProcessParIDGet.Error THEN
			// Transfer error id, reset funtion block, reset command
			IF AxisParId.ErrId = 0 THEN
				AxisParId.ErrId := AxisParIdInternal.ProcessParIDGet.ErrorID;
			END_IF

			FOR AxisParIdInternal.n:=1 TO AxisParNum DO
				FOR AxisParIdInternal.m:=1 TO AxisParIdInternal.DataOnceGetIdx DO
					IF AxisParIdInternal.DataOnceGet[AxisParIdInternal.m].ParID = AxisParId.ParIds[AxisParIdInternal.n].ParID AND AxisParIdInternal.DataOnceGet[AxisParIdInternal.m].VariableAddress = AxisParIdInternal.McVariableAdr[AxisParIdInternal.n] THEN
						AxisParId.ParIds[AxisParIdInternal.n].Execute := mcACPAX_PARID_DONE;
					END_IF
				END_FOR;
			END_FOR;
			brsmemset(ADR(AxisParIdInternal.DataOnceGet), 0, SIZEOF(AxisParIdInternal.DataOnceGet));
			AxisParIdInternal.DataOnceGetIdx := 0;

			AxisParIdInternal.ProcessParIDGet.Execute := 0;
		END_IF
	END_IF

	// --------------------------------------------------------------------------
	// Create set once queue
	IF AxisParIdInternal.DataOnceSetIdx = 0  THEN
		FOR AxisParIdInternal.n:=1 TO AxisParNum DO
			// Transfer set once data
			IF AxisParId.ParIds[AxisParIdInternal.n].Execute = mcACPAX_PARID_SET_ONCE THEN
				AxisParIdInternal.DataOnceSetIdx := AxisParIdInternal.DataOnceSetIdx + 1;
				GetVarData;
				// Variable data is valid
				IF AxisParIdInternal.VariableStatus = 0 THEN
					AxisParIdInternal.DataOnceSet[AxisParIdInternal.DataOnceSetIdx].ParID := AxisParId.ParIds[AxisParIdInternal.n].ParID;
					AxisParIdInternal.DataOnceSet[AxisParIdInternal.DataOnceSetIdx].VariableAddress := AxisParIdInternal.McVariableAdr[AxisParIdInternal.n];
					AxisParIdInternal.DataOnceSet[AxisParIdInternal.DataOnceSetIdx].DataType := AxisParIdInternal.McVariableType[AxisParIdInternal.n];
				// Error reading variable data
				ELSE
					AxisParId.ErrId := AxisParIdInternal.VariableStatus;
					AxisParId.ParIds[AxisParIdInternal.n].Execute := mcACPAX_PARID_DONE;
				END_IF

			END_IF
		END_FOR;
	END_IF

	// --------------------------------------------------------------------------
	// Execute set once queue
	IF AxisParIdInternal.DataOnceSetIdx > 0 THEN
		// Preset function block
		AxisParIdInternal.ProcessParIDSet.Execute := 1;
		AxisParIdInternal.ProcessParIDSet.Axis := AxisParId.MpLink;
		AxisParIdInternal.ProcessParIDSet.DataAddress := ADR(AxisParIdInternal.DataOnceSet);
		AxisParIdInternal.ProcessParIDSet.NumberOfParIDs := AxisParIdInternal.DataOnceSetIdx;
		AxisParIdInternal.ProcessParIDSet.Mode := mcACPAX_PARID_SET;

		// Finish when done
		IF AxisParIdInternal.ProcessParIDSet.Done OR AxisParIdInternal.ProcessParIDSet.Error THEN
			// Transfer error id, reset funtion block, reset command
			IF AxisParId.ErrId = 0 THEN
				AxisParId.ErrId := AxisParIdInternal.ProcessParIDSet.ErrorID;
			END_IF

			FOR AxisParIdInternal.n:=1 TO AxisParNum DO
				FOR AxisParIdInternal.m:=1 TO AxisParIdInternal.DataOnceSetIdx DO
					IF AxisParIdInternal.DataOnceSet[AxisParIdInternal.m].ParID = AxisParId.ParIds[AxisParIdInternal.n].ParID AND AxisParIdInternal.DataOnceSet[AxisParIdInternal.m].VariableAddress = AxisParIdInternal.McVariableAdr[AxisParIdInternal.n] THEN
						AxisParId.ParIds[AxisParIdInternal.n].Execute := mcACPAX_PARID_DONE;
					END_IF
				END_FOR;
			END_FOR;
			brsmemset(ADR(AxisParIdInternal.DataOnceSet), 0, SIZEOF(AxisParIdInternal.DataOnceSet));
			AxisParIdInternal.DataOnceSetIdx := 0;

			AxisParIdInternal.ProcessParIDSet.Execute := 0;
		END_IF
	END_IF

	// --------------------------------------------------------------------------
	// Create get cylcic queue
	IF EDGEPOS(AxisParId.CmdUpdate) THEN
		// Create new queue
		FOR AxisParIdInternal.n:=1 TO AxisParNum DO
			// Transfer get cyclic data
			IF AxisParId.ParIds[AxisParIdInternal.n].Execute = mcACPAX_PARID_GET_CYCLIC OR AxisParId.ParIds[AxisParIdInternal.n].Execute = mcACPAX_PARID_GET_MULTI THEN
				AxisParIdInternal.DataCyclicGetIdx := AxisParIdInternal.DataCyclicGetIdx + 1;
				GetVarData;
				// Variable data is valid
				IF AxisParIdInternal.VariableStatus = 0 THEN
					AxisParIdInternal.DataCylicGet[AxisParIdInternal.DataCyclicGetIdx].ParID := AxisParId.ParIds[AxisParIdInternal.n].ParID;
					AxisParIdInternal.DataCylicGet[AxisParIdInternal.DataCyclicGetIdx].VariableAddress := AxisParIdInternal.McVariableAdr[AxisParIdInternal.n];
					AxisParIdInternal.DataCylicGet[AxisParIdInternal.DataCyclicGetIdx].DataType := AxisParIdInternal.McVariableType[AxisParIdInternal.n];
					IF AxisParId.ParIds[AxisParIdInternal.n].Execute = mcACPAX_PARID_GET_CYCLIC THEN
						AxisParIdInternal.DataCylicGet[AxisParIdInternal.DataCyclicGetIdx].RefreshMode := mcACPAX_CYCLIC_EVERY_RECORD;
					ELSE
						AxisParIdInternal.DataCylicGet[AxisParIdInternal.DataCyclicGetIdx].RefreshMode := mcACPAX_CYCLIC_MULTIPLEXED;
					END_IF
				// Error reading variable data
				ELSE
					AxisParId.ErrId := AxisParIdInternal.VariableStatus;
					AxisParId.ParIds[AxisParIdInternal.n].Execute := mcACPAX_PARID_DONE;
				END_IF
			END_IF
		END_FOR;
	END_IF

	// --------------------------------------------------------------------------
	// Create set cylcic queue
	IF EDGEPOS(AxisParId.CmdUpdate) THEN
		// Create new queue
		FOR AxisParIdInternal.n:=1 TO AxisParNum DO
			// Transfer set cyclic data
			IF AxisParId.ParIds[AxisParIdInternal.n].Execute = mcACPAX_PARID_SET_CYCLIC OR AxisParId.ParIds[AxisParIdInternal.n].Execute = mcACPAX_PARID_SET_MULTI THEN
				AxisParIdInternal.DataCyclicSetIdx := AxisParIdInternal.DataCyclicSetIdx + 1;
				GetVarData;
				// Variable data is valid
				IF AxisParIdInternal.VariableStatus = 0 THEN
					AxisParIdInternal.DataCylicSet[AxisParIdInternal.DataCyclicSetIdx].ParID := AxisParId.ParIds[AxisParIdInternal.n].ParID;
					AxisParIdInternal.DataCylicSet[AxisParIdInternal.DataCyclicSetIdx].VariableAddress := AxisParIdInternal.McVariableAdr[AxisParIdInternal.n];
					AxisParIdInternal.DataCylicSet[AxisParIdInternal.DataCyclicSetIdx].DataType := AxisParIdInternal.McVariableType[AxisParIdInternal.n];
					IF AxisParId.ParIds[AxisParIdInternal.n].Execute = mcACPAX_PARID_SET_CYCLIC THEN
						AxisParIdInternal.DataCylicSet[AxisParIdInternal.DataCyclicSetIdx].RefreshMode := mcACPAX_CYCLIC_EVERY_RECORD;
					ELSE
						AxisParIdInternal.DataCylicSet[AxisParIdInternal.DataCyclicSetIdx].RefreshMode := mcACPAX_CYCLIC_MULTIPLEXED;
					END_IF
				// Error reading variable data
				ELSE
					AxisParId.ErrId := AxisParIdInternal.VariableStatus;
					AxisParId.ParIds[AxisParIdInternal.n].Execute := mcACPAX_PARID_DONE;
				END_IF

			END_IF
		END_FOR;
	END_IF

	// --------------------------------------------------------------------------
	// Execute set cyclic queue
	IF AxisParIdInternal.DataCyclicSetIdx > 0 THEN
		// Preset function block
		AxisParIdInternal.CyclicProcessParIDSet.Enable := TRUE;
		AxisParIdInternal.CyclicProcessParIDSet.Axis := AxisParId.MpLink;
		AxisParIdInternal.CyclicProcessParIDSet.DataAddress := ADR(AxisParIdInternal.DataCylicSet);
		AxisParIdInternal.CyclicProcessParIDSet.NumberOfParIDs := AxisParIdInternal.DataCyclicSetIdx;
		AxisParIdInternal.CyclicProcessParIDSet.Mode := mcACPAX_CYCLIC_PARID_WRITE;

		// Log error
		IF AxisParIdInternal.CyclicProcessParIDSet.Error AND AxisParId.ErrId = 0 THEN
			AxisParId.ErrId := AxisParIdInternal.CyclicProcessParIDSet.ErrorID;
		END_IF
	ELSE
		AxisParIdInternal.CyclicProcessParIDSet.Enable := FALSE;
	END_IF

	// Cyclic function calls
	AxisParIdInternal.ProcessParIDGet();
	AxisParIdInternal.ProcessParIDSet();
	AxisParIdInternal.CyclicProcessParIDGet();
	AxisParIdInternal.CyclicProcessParIDSet();

	// --------------------------------------------------------------------------
	// Execute get cyclic queue
	IF AxisParIdInternal.DataCyclicGetIdx > 0 THEN
		// Preset function block
		AxisParIdInternal.CyclicProcessParIDGet.Enable := TRUE;
		AxisParIdInternal.CyclicProcessParIDGet.Axis := AxisParId.MpLink;
		AxisParIdInternal.CyclicProcessParIDGet.DataAddress := ADR(AxisParIdInternal.DataCylicGet);
		AxisParIdInternal.CyclicProcessParIDGet.NumberOfParIDs := AxisParIdInternal.DataCyclicGetIdx;
		AxisParIdInternal.CyclicProcessParIDGet.Mode := mcACPAX_CYCLIC_PARID_READ;

		// Log error
		IF AxisParIdInternal.CyclicProcessParIDGet.Error AND AxisParId.ErrId = 0 THEN
			AxisParId.ErrId := AxisParIdInternal.CyclicProcessParIDGet.ErrorID;
		END_IF
	ELSE
		AxisParIdInternal.CyclicProcessParIDGet.Enable := FALSE;
	END_IF

	// --------------------------------------------------------------------------
	// Get cyclic pard id information
	IF AxisParId.CmdUpdate AND (AxisParIdInternal.DataCyclicGetIdx > 0 AND AxisParIdInternal.CyclicProcessParIDGet.Valid OR AxisParIdInternal.DataCyclicGetIdx = 0) AND (AxisParIdInternal.DataCyclicSetIdx > 0 AND AxisParIdInternal.CyclicProcessParIDSet.Valid  OR AxisParIdInternal.DataCyclicSetIdx = 0) THEN
		// Preset function block
		AxisParIdInternal.GetCyclicDataInfo.Execute := TRUE;
		AxisParIdInternal.GetCyclicDataInfo.Axis := AxisParId.MpLink;

		// Finish when done
		IF AxisParIdInternal.GetCyclicDataInfo.Done OR AxisParIdInternal.GetCyclicDataInfo.Error THEN
			// Transfer error id, reset funtion block, reset command
			IF AxisParId.ErrId = 0 THEN
				AxisParId.ErrId := AxisParIdInternal.GetCyclicDataInfo.ErrorID;
			END_IF

			// Transfer bytes used
			AxisParId.MaxWriteDataBytes := AxisParIdInternal.GetCyclicDataInfo.CyclicDataInfo.Write.Record.Size;
			AxisParId.MaxReadDataBytes := 0;
			IF AxisParIdInternal.GetCyclicDataInfo.CyclicDataInfo.Read.RecordCount > 0 THEN
				FOR AxisParIdInternal.m:=0 TO AxisParIdInternal.GetCyclicDataInfo.CyclicDataInfo.Read.RecordCount - 1 DO
					IF AxisParIdInternal.GetCyclicDataInfo.CyclicDataInfo.Read.Record[AxisParIdInternal.m].Size > AxisParId.MaxReadDataBytes THEN
						AxisParId.MaxReadDataBytes := AxisParIdInternal.GetCyclicDataInfo.CyclicDataInfo.Read.Record[AxisParIdInternal.m].Size;
					END_IF
				END_FOR;
			END_IF

			AxisParId.CmdUpdate := 0;
		END_IF
		AxisParIdInternal.GetCyclicDataInfo();
	END_IF

END_ACTION

// --------------------------------------------------------------------------
// Get variable details
ACTION GetVarData:
	// Get variable address
	AxisParIdInternal.VariableStatus := PV_xgetadr(ADR(AxisParId.ParIds[AxisParIdInternal.n].Variable), ADR(AxisParIdInternal.VariableAdr), ADR(AxisParIdInternal.VariableLen));
	IF AxisParIdInternal.VariableStatus = 0 THEN
		// Get variable data type
		AxisParIdInternal.VariableStatus := PV_ninfo(ADR(AxisParId.ParIds[AxisParIdInternal.n].Variable), ADR(AxisParIdInternal.VariableType), ADR(AxisParIdInternal.VariableLen), ADR(AxisParIdInternal.VariableDimension));
		IF AxisParIdInternal.VariableStatus = 0 THEN
			// Transfer address and translate variable type to mc type
			AxisParIdInternal.McVariableAdr[AxisParIdInternal.n] := AxisParIdInternal.VariableAdr;
			// If variable if structure or array, use void
			IF AxisParIdInternal.VariableDimension > 1 THEN
				AxisParIdInternal.McVariableType[AxisParIdInternal.n] := mcACPAX_PARTYPE_VOID;
				// Assign type for standard types
			ELSE
				CASE AxisParIdInternal.VariableType OF
					SYSLIB_IEC_TYPE_BOOL:
			  			AxisParIdInternal.McVariableType[AxisParIdInternal.n] := mcACPAX_PARTYPE_BOOL;
					SYSLIB_IEC_TYPE_REAL:
						AxisParIdInternal.McVariableType[AxisParIdInternal.n] := mcACPAX_PARTYPE_REAL;
					SYSLIB_IEC_TYPE_SINT:
						AxisParIdInternal.McVariableType[AxisParIdInternal.n] := mcACPAX_PARTYPE_SINT;
					SYSLIB_IEC_TYPE_USINT:
						AxisParIdInternal.McVariableType[AxisParIdInternal.n] := mcACPAX_PARTYPE_USINT;
					SYSLIB_IEC_TYPE_INT:
						AxisParIdInternal.McVariableType[AxisParIdInternal.n] := mcACPAX_PARTYPE_INT;
					SYSLIB_IEC_TYPE_UINT:
						AxisParIdInternal.McVariableType[AxisParIdInternal.n] := mcACPAX_PARTYPE_UINT;
					SYSLIB_IEC_TYPE_DINT:
						AxisParIdInternal.McVariableType[AxisParIdInternal.n] := mcACPAX_PARTYPE_DINT;
					SYSLIB_IEC_TYPE_UDINT:
						AxisParIdInternal.McVariableType[AxisParIdInternal.n] := mcACPAX_PARTYPE_UDINT;
					ELSE
						AxisParIdInternal.McVariableType[AxisParIdInternal.n] := mcACPAX_PARTYPE_VOID;
				END_CASE;
			END_IF
		ELSE
			IF AxisParId.ErrId = 0 THEN
				AxisParId.ErrId := AxisParIdInternal.VariableStatus;
			END_IF
		END_IF
	ELSE
		IF AxisParId.ErrId = 0 THEN
			AxisParId.ErrId := AxisParIdInternal.VariableStatus;
		END_IF
	END_IF
END_ACTION
```

#### revision.txt
```
Version 5
- Update to mappMotion 5.22.1
- Improved error handling

Version 4
- Removed dependency from common
- Added cyclic par id exchange
- Simplified interface

Version 3
- Renamed function block

Version 2
- Renamed action

Version 1
- First release
```

### Program Logical/axis_1 (IEC)

#### Main.st - Init, cyclic, exit code
```iecst
PROGRAM _INIT
	// --------------------------------------------------------------------------
	// Set standard motion parameters
	MpAxisBasicPar.Acceleration := 10000;
	MpAxisBasicPar.Deceleration := 10000;
	MpAxisBasicPar.Stop.Deceleration := 10000;
	MpAxisBasicPar.Velocity := 500;

	// --------------------------------------------------------------------------
	// Set brake parameters, disable brake restrictions
	AxisBrake.ParAxis := gAxis_1;
	AxisBrake.ParBrake.RestrictedBrakeControl := mcSWITCH_OFF;
	AxisBrake.CmdSetPar := TRUE;

	// --------------------------------------------------------------------------
	// Acknoledge encoder battery error
	mcACPAX_UDINT[1] := 1;
	AxisParId.ParAxis := gAxis_1;
	AxisParId.ParNum := 1;
	AxisParId.ParIds[1].ParID := 719;
	AxisParId.ParIds[1].VariableAddress := ADR(mcACPAX_UDINT);
	AxisParId.ParIds[1].DataType := mcACPAX_PARTYPE_UDINT;
	AxisParId.CmdSetPar := TRUE;

END_PROGRAM

PROGRAM _CYCLIC

	// --------------------------------------------------------------------------
	// Call axis main function block
	MpAxisBasic_1.Enable := 1;
	MpAxisBasic_1.MpLink := ADR(gAxis_1);
	MpAxisBasic_1.Parameters := ADR(MpAxisBasicPar);
	MpAxisBasic_1();

	// --------------------------------------------------------------------------
	// Call axis actions used for this drive
	Brake;
	ParID;

END_PROGRAM

PROGRAM _EXIT
	(* Insert code here *)

END_PROGRAM
```

#### Variables.var - Local variables
```iecst
VAR
	MpAxisBasic_1 : MpAxisBasic;
	MpAxisBasicPar : MpAxisBasicParType;
	mcACPAX_UDINT : UDINT;
	mcSPEED_MAX : DINT;
	mcSPEED_ACTUAL : REAL;
END_VAR
```

- AxisProtoBrake.st (reference to Logical/AxisProto/AxisProtoBrake.st)

- AxisProtoBrake.typ (reference to Logical/AxisProto/AxisProtoBrake.typ)

- AxisProtoBrake.var (reference to Logical/AxisProto/AxisProtoBrake.var)

- AxisProtoParId.st (reference to Logical/AxisProto/AxisProtoParId.st)

- AxisProtoParId.typ (reference to Logical/AxisProto/AxisProtoParId.typ)

- AxisProtoParId.var (reference to Logical/AxisProto/AxisProtoParId.var)

### Program Logical/Axis_2 (IEC)

#### Main.st - Init, cyclic, exit code
```iecst
PROGRAM _INIT
	// --------------------------------------------------------------------------
	// Set brake parameters, disable brake restrictions
	AxisBrake.ParAxis := gAxis_2;
	AxisBrake.ParBrake.RestrictedBrakeControl := mcSWITCH_OFF;
	AxisBrake.CmdSetPar := TRUE;

	// --------------------------------------------------------------------------
	// Acknoledge encoder battery error
	mcACPAX_UDINT[1] := 1;
	AxisParId.ParAxis := gAxis_2;
	AxisParId.ParNum := 1;
	AxisParId.ParIds[1].ParID := 719;
	AxisParId.ParIds[1].VariableAddress := ADR(mcACPAX_UDINT);
	AxisParId.ParIds[1].DataType := mcACPAX_PARTYPE_UDINT;
	AxisParId.CmdSetPar := TRUE;

END_PROGRAM

PROGRAM _CYCLIC
	// --------------------------------------------------------------------------
	// Call axis main function block
	MpAxisBasic_1.Enable := 1;
	MpAxisBasic_1.MpLink := ADR(gAxis_2);
	MpAxisBasic_1.Parameters := ADR(MpAxisBasicPar);
	MpAxisBasic_1();

	// --------------------------------------------------------------------------
	// Call axis actions used for this drive
	Brake;
	ParID;

END_PROGRAM

PROGRAM _EXIT
	(* Insert code here *)

END_PROGRAM
```

#### Variables.var - Local variables
```iecst
VAR
	MpAxisBasic_1 : MpAxisBasic;
	MpAxisBasicPar : MpAxisBasicParType;
END_VAR
```

- AxisProtoBrake.st (reference to Logical/AxisProto/AxisProtoBrake.st)

- AxisProtoBrake.typ (reference to Logical/AxisProto/AxisProtoBrake.typ)

- AxisProtoBrake.var (reference to Logical/AxisProto/AxisProtoBrake.var)

- AxisProtoParId.st (reference to Logical/AxisProto/AxisProtoParId.st)

- AxisProtoParId.typ (reference to Logical/AxisProto/AxisProtoParId.typ)

- AxisProtoParId.var (reference to Logical/AxisProto/AxisProtoParId.var)

- Visualisation Logical/mappView (not shown)

Listed in the project but not available here: Logical/Global.typ, Logical/Global.var, Logical/AxisProto/General/AxisProtoGlobal.typ, Logical/axis_1/Types.typ, Logical/Axis_2/Types.typ, Logical/AxisProto/AxisProtoGlobal.typ, Logical/AxisProto/AxisProtoGlobal.var
